FUNCTION_BLOCK LimitOutput
VAR_INPUT
	IN: LREAL;
	LIM: LREAL;
	LIM_FB: LREAL;
	T: TIME := T#60S;
END_VAR
VAR_OUTPUT
	OUT: LREAL;
END_VAR
VAR
	TempIN: LREAL;
	TempOut: LREAL;
	Sum: LREAL;
	Timer: Timer;
	Delta: LREAL;
	d: LINT;
	FirstTime: bool;
END_VAR

IF NOT FirstTime THEN
	FirstTime := TRUE;
	d := TO_LINT(T);
	IF d > 0 THEN
		Delta := 1000.0 / TO_LREAL(d);
	ELSE
		Delta := 0.01;	
	END_IF
END_IF

TempIN := IN;

IF Timer.ElapsedTime() > 1000 THEN	
	IF LIM_FB > LIM AND Sum > 0 THEN
		Sum := Sum - Delta;
		IF Sum < 0 THEN
			Sum := 0;
		END_IF
	END_IF
	IF LIM_FB < LIM AND Sum < 1 THEN
		Sum := Sum + Delta;
		IF Sum > 1 THEN
			Sum := 1;
		END_IF
	END_IF
	Timer.Restart();
END_IF
TempOut := TempIN - Sum;
IF TempOut < 0 THEN
	TempOut := 0;
END_IF
IF TempOut > 1 THEN
	TempOut := 1;
END_IF
OUT := TempOut;

END_FUNCTION_BLOCK

(* stored: Version 1.1.0.1, ProductVersion 3.1.4024.6
   POU LimitOutput: Id {8ae27181-a104-4ac6-aeea-42c26e637f82}, SpecialFunc None *)
